Universal Robots PolyScope program: SandCube2.urp

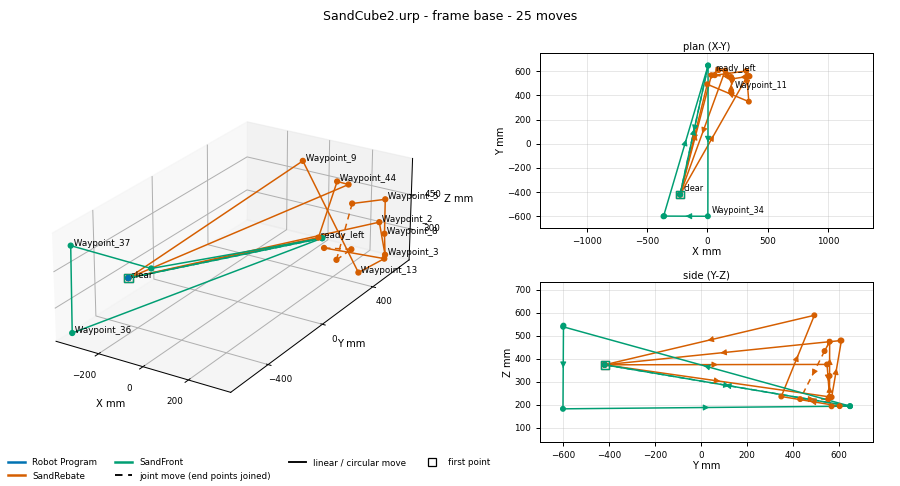
[picture p0: tool path of SandCube2.urp in frame base, 25 of 25 moves have a stored position in this frame; points joined in program order, loops and branches not executed]
Program SandCube2 (installation=main2 directory=/programs createdIn=5.11.5.1010327 lastSavedIn=5.11.5.1010327 robotSerialNumber=20215500677)
Calibrated DH parameters: a=[0.000204, -0.239222, -0.391845, -0.000001, 0.000022, 0]; d=[0.162722, -355.808559, 353.37206, 2.570385, 0.099741, 0.099629]; alpha=[1.571124, 0.000988, 0.008295, 1.568963, -1.570303, 0]; deltaTheta=[0, -0.973091, 7.204745, 0.05153, 0, 0]
Robot Program (runOnlyOnce=false)
  Folder Main
    MoveJ speed 60 deg/s, acceleration 80 deg/s^2 (useActiveTCP=false) tcp=DynabradeDual; feature=CubeFront
      Waypoint clear: TCP in base x=-225.713 y=-419.127 z=372.802 mm, rx=0.1834 ry=-2.2071 rz=2.1997 rad; joints [13.855, -106.476, 145.256, -123.976, 44.893, -104.552] deg; TCP offset x=3.18 y=114.64 z=98.2 mm, rx=-0.7854 ry=0 rz=0 rad; feature pose in base x=2.048 y=-607.004 z=173.227 mm, rx=-0.0204 ry=-2.2235 rz=-2.2094 rad
      URCap Zero FT Sensor (Robotiq_Copilot, Robotiq Inc.) dataModel(NodeInitializedKey=true, WaitForSteadyWrenchOptionKey=true)
    CubeFront := CubeFront
    Call SandFront
    CubeFront := SandBack
    Call SandFront
    SuppressedNode
      Call SprayFront
    SuppressedNode
      Call SprayFront
  SuppressedNode
    Folder Chamfer
      MoveL speed 250 mm/s, acceleration 1200 mm/s^2 (useActiveTCP=true) feature=Base
        MoveJ speed 60 deg/s, acceleration 80 deg/s^2 (useActiveTCP=true) feature=CubeFront
          Waypoint Waypoint_14: TCP in base x=40.557 y=344.633 z=644.318 mm, rx=1.3155 ry=-1.3725 rz=-1.2523 rad; joints [213.145, -95.792, 65.461, -31.373, -65.462, -328.995] deg; feature pose in base x=6.058 y=653.089 z=192.929 mm, rx=1.5716 ry=0.003 rz=-0.0025 rad
          Waypoint Waypoint_15: TCP in base x=-6.602 y=417.802 z=666.352 mm, rx=-2.8064 ry=0.3635 rz=0.257 rad; joints [242.083, -106.85, 75.59, -118.753, -70.655, -356.384] deg
          Waypoint Waypoint_16: TCP in base x=7.321 y=653.157 z=552.583 mm, rx=-2.3553 ry=0.0014 rz=0.0042 rad; joints [252.243, -84.14, 86.654, -182.715, -72.191, -359.211] deg
        URCap Find Surface (Robotiq_Copilot, Robotiq Inc.) dataModel(NodeInitializedKey=true, ZeroSensorBeforeKey=true, WaitForSteadyWrenchOptionKey=false, ls_force=10.0, ls_distance=100.0, ls_speed=5.0, ls_if_distance=false, ls_if_force=false); state(isChildrenLocked=true)
          'Add Stop conditions from the Find Surface node'
        URCap Finishing Tool Control (Robotiq_Copilot, Robotiq Inc.) dataModel(ToolOutputNameKey=digital_out[0], HackTriggeringContributionIsDefinedMethodKey=true)
        Wait Sleep waitTime=0.5
        MoveDirectionNode (selectedDirection=XPlus toolParams=0.15, 1.2) feature(featureName=CubeFront)
          Until DISTANCE (allowActions=false deceleration=3 distanceNodeType=STOP) Distance=0.35; motionParameters(blendRadius=0)
        MoveDirectionNode (selectedDirection=ZMinus) feature=Joint_6_name
          Until DISTANCE (allowActions=false deceleration=3 distanceNodeType=STOP) Distance=0.025; motionParameters(blendRadius=0)
        URCap Finishing Tool Control (Robotiq_Copilot, Robotiq Inc.) dataModel(FinishingToolStateKey=false, ToolOutputNameKey=digital_out[0], HackTriggeringContributionIsDefinedMethodKey=true)
        Waypoint Waypoint_18: TCP in base x=366.179 y=605.982 z=520.828 mm, rx=-1.6861 ry=0.1385 rz=1.2496 rad; joints [208.374, -44.818, 51.064, -237.69, -37.068, -253.683] deg
        URCap Find Surface (Robotiq_Copilot, Robotiq Inc.) dataModel(NodeInitializedKey=true, ZeroSensorBeforeKey=true, WaitForSteadyWrenchOptionKey=false, ls_force=10.0, ls_distance=100.0, ls_speed=5.0, ls_if_distance=false, ls_if_force=false); state(isChildrenLocked=true)
          'Add Stop conditions from the Find Surface node'
        URCap Finishing Tool Control (Robotiq_Copilot, Robotiq Inc.) dataModel(ToolOutputNameKey=digital_out[0], HackTriggeringContributionIsDefinedMethodKey=true)
        MoveDirectionNode (selectedDirection=YMinus toolParams=0.15, 1.2) feature(featureName=CubeFront)
          Until DISTANCE (allowActions=false deceleration=3 distanceNodeType=STOP) Distance=0.35; motionParameters(blendRadius=0)
        URCap Finishing Tool Control (Robotiq_Copilot, Robotiq Inc.) dataModel(FinishingToolStateKey=false, ToolOutputNameKey=digital_out[0], HackTriggeringContributionIsDefinedMethodKey=true)
        MoveDirectionNode (selectedDirection=ZMinus) feature=Joint_6_name
          Until DISTANCE (allowActions=false deceleration=3 distanceNodeType=STOP) Distance=0.05; motionParameters(blendRadius=0)
        Waypoint Waypoint_20: TCP in base x=366.722 y=626.869 z=194.22 mm, rx=-1.1174 ry=-0.6786 rz=-0.9417 rad; joints [212.764, -30.352, 68.609, -330.279, -35.41, -327.866] deg
        URCap Find Surface (Robotiq_Copilot, Robotiq Inc.) dataModel(NodeInitializedKey=true, ZeroSensorBeforeKey=true, WaitForSteadyWrenchOptionKey=false, ls_force=10.0, ls_distance=100.0, ls_speed=5.0, ls_if_distance=false, ls_if_force=false); state(isChildrenLocked=true)
          'Add Stop conditions from the Find Surface node'
        URCap Finishing Tool Control (Robotiq_Copilot, Robotiq Inc.) dataModel(ToolOutputNameKey=digital_out[0], HackTriggeringContributionIsDefinedMethodKey=true)
        Waypoint Waypoint_19: motionParameters(jointSpeed=1.047198 jointAcceleration=1.396263 cartesianSpeed=0.05 cartesianAcceleration=1.2); TCP in base x=29.784 y=640.794 z=212.679 mm, rx=-1.2502 ry=-0.1072 rz=-0.0765 rad; joints [247.483, -34.268, 98.117, -310.948, -74.468, -342.493] deg
        URCap Finishing Tool Control (Robotiq_Copilot, Robotiq Inc.) dataModel(FinishingToolStateKey=false, ToolOutputNameKey=digital_out[0], HackTriggeringContributionIsDefinedMethodKey=true)
        MoveDirectionNode (selectedDirection=ZMinus) feature=Joint_6_name
          Until DISTANCE (allowActions=false deceleration=3 distanceNodeType=STOP) Distance=0.05; motionParameters(blendRadius=0)
Event  expression=digital_in[1]≠ True
  Set DigitalOutput pin=digital_out[0]; digitalValue=0
  Set DigitalOutput pin=digital_out[1]; digitalValue=0
  Halt
SubProgram SandRebate (keepSynchronizedWithDisk=false)
  Folder sandRebate
    MoveJ speed 60 deg/s, acceleration 80 deg/s^2 (useActiveTCP=false) tcp=DynabradeDual; feature=CubeFront
      Waypoint clear: TCP in base x=-225.713 y=-419.127 z=372.802 mm, rx=0.1834 ry=-2.2071 rz=2.1997 rad; joints [13.855, -106.476, 145.256, -123.976, 44.893, -104.552] deg; feature pose in base x=2.048 y=-607.004 z=173.227 mm, rx=-0.0204 ry=-2.2235 rz=-2.2094 rad
      URCap Zero FT Sensor (Robotiq_Copilot, Robotiq Inc.) dataModel(NodeInitializedKey=true, WaitForSteadyWrenchOptionKey=true)
      MoveL speed 250 mm/s, acceleration 1200 mm/s^2 (useActiveTCP=false) tcp=DynabradeDual; feature=CubeFront
        Waypoint ready_left: TCP in base x=33.773 y=568.14 z=232.075 mm, rx=-1.2213 ry=-1.2022 rz=1.1979 rad; joints [233.005, -43.676, 101.374, -178.142, 55.004, -44.435] deg; TCP offset x=3.18 y=114.64 z=98.2 mm, rx=-0.7854 ry=0 rz=0 rad; feature pose in base x=9.685 y=618.378 z=176.869 mm, rx=1.5687 ry=-0.014 rz=-0.0074 rad
        URCap Find Surface (Robotiq_Copilot, Robotiq Inc.) dataModel(NodeInitializedKey=true, WaitForSteadyWrenchOptionKey=false, ls_force=10.0, ls_distance=100.0, ls_speed=5.0, ZeroSensorBeforeKey=true, ls_if_distance=false, ls_if_force=false); state(isChildrenLocked=true)
          'Add Stop conditions from the Find Surface node'
        URCap Finishing Tool Control (Robotiq_Copilot, Robotiq Inc.) dataModel(ToolOutputNameKey=digital_out[0], HackTriggeringContributionIsDefinedMethodKey=true)
        Wait Sleep waitTime=0.5
        Force Simple feature=Joint_6_name; selection=[0, 0, 1, 0, 0, 0]; wrench=[0, 0, 5, 0, 0, 0]; limitsForce=[0.15, 0.15, 0.15, 1.047198, 1.047198, 1.047198]; limitsMotion=[0.1, 0.1, 0.1, 0.349066, 0.349066, 0.349066]
          Waypoint Waypoint_44: motionParameters(jointSpeed=1.047198 jointAcceleration=1.396263 cartesianSpeed=0.05 cartesianAcceleration=1.2); TCP in base x=92.634 y=610.628 z=478.238 mm, rx=-0.8396 ry=-1.4025 rz=0.8393 rad; joints [232.816, -51.553, 73.036, -159.375, 69.035, -55.707] deg; TCP offset x=3.18 y=114.64 z=98.2 mm, rx=-0.7854 ry=0 rz=0 rad; feature pose in base x=85.344 y=655.608 z=190.328 mm, rx=1.5707 ry=0.001 rz=-0.0012 rad
        URCap Finishing Tool Control (Robotiq_Copilot, Robotiq Inc.) dataModel(ToolOutputNameKey=digital_out[0], HackTriggeringContributionIsDefinedMethodKey=true, FinishingToolStateKey=false)
        Waypoint Waypoint_4: TCP in base x=147.72 y=606.874 z=478.224 mm, rx=-0.8396 ry=-1.4025 rz=0.8394 rad; joints [229.161, -48.232, 67.407, -157.963, 71.791, -53.121] deg
        Waypoint clear: TCP in base x=-225.713 y=-419.127 z=372.802 mm, rx=0.1834 ry=-2.2071 rz=2.1997 rad; joints [13.855, -106.476, 145.256, -123.976, 44.893, -104.552] deg; feature pose in base x=2.048 y=-607.004 z=173.227 mm, rx=-0.0204 ry=-2.2235 rz=-2.2094 rad
        Waypoint Waypoint_2: TCP in base x=324.212 y=548.214 z=374.491 mm, rx=-1.2092 ry=1.2092 rz=-1.2092 rad; joints [245.591, -72.937, 106.11, -100.873, 130.52, -237.51] deg; feature pose in base x=6.058 y=653.089 z=192.929 mm, rx=1.5716 ry=0.003 rz=-0.0025 rad
        Waypoint Waypoint_3: TCP in base x=348.673 y=558.868 z=233.4 mm, rx=-1.199 ry=1.2125 rz=-1.2251 rad; joints [243.834, -57.283, 109.058, -119.037, 129.688, -236.76] deg; TCP offset x=3.18 y=114.64 z=98.2 mm, rx=-0.7854 ry=0 rz=0 rad; feature pose in base x=9.685 y=618.378 z=176.869 mm, rx=1.5687 ry=-0.014 rz=-0.0074 rad
        URCap Find Surface (Robotiq_Copilot, Robotiq Inc.) dataModel(NodeInitializedKey=true, WaitForSteadyWrenchOptionKey=false, ls_force=10.0, ls_distance=100.0, ls_speed=5.0, ZeroSensorBeforeKey=true, ls_if_distance=false, ls_if_force=false); state(isChildrenLocked=true)
          'Add Stop conditions from the Find Surface node'
        URCap Finishing Tool Control (Robotiq_Copilot, Robotiq Inc.) dataModel(ToolOutputNameKey=digital_out[0], HackTriggeringContributionIsDefinedMethodKey=true)
        Wait Sleep waitTime=0.5
        Force Simple feature=Joint_6_name; selection=[0, 0, 1, 0, 0, 0]; wrench=[0, 0, 5, 0, 0, 0]; limitsForce=[0.15, 0.15, 0.15, 1.047198, 1.047198, 1.047198]; limitsMotion=[0.1, 0.1, 0.1, 0.349066, 0.349066, 0.349066]
          Waypoint Waypoint_8: motionParameters(jointSpeed=1.047198 jointAcceleration=1.396263 cartesianSpeed=0.05 cartesianAcceleration=1.2); TCP in base x=343.269 y=559.127 z=324.456 mm, rx=2.2046 ry=-0.0122 rz=2.2215 rad; joints [241.547, -71.33, 93.008, -21.809, 107.451, -270.149] deg; TCP offset x=3.18 y=114.64 z=98.2 mm, rx=-0.7854 ry=0 rz=0 rad
          Waypoint Waypoint_5: motionParameters(jointSpeed=1.047198 jointAcceleration=1.396263 cartesianSpeed=0.05 cartesianAcceleration=1.2); TCP in base x=342.13 y=559.447 z=473.527 mm, rx=2.1002 ry=0.2016 rz=2.1132 rad; joints [241.727, -73.096, 71.489, 10.077, 107.843, -275.731] deg; TCP offset x=3.18 y=114.64 z=98.2 mm, rx=-0.7854 ry=0 rz=0 rad
        URCap Finishing Tool Control (Robotiq_Copilot, Robotiq Inc.) dataModel(FinishingToolStateKey=false, ToolOutputNameKey=digital_out[0], HackTriggeringContributionIsDefinedMethodKey=true)
        Waypoint Waypoint_17: TCP in base x=204.615 y=537.314 z=432.533 mm, rx=-1.1836 ry=-1.1482 rz=-1.3158 rad; joints [212.134, -87.867, 98.846, 1.992, -9.504, -287.219] deg; TCP offset x=3.18 y=114.64 z=98.2 mm, rx=-0.7854 ry=0 rz=0 rad; feature pose in base x=6.058 y=653.089 z=192.929 mm, rx=1.5716 ry=0.003 rz=-0.0025 rad
        MoveJ speed 60 deg/s, acceleration 80 deg/s^2 (useActiveTCP=true) feature=CubeFront
          Waypoint Waypoint_11: TCP in base x=197.023 y=431.256 z=223.624 mm, rx=2.362 ry=2.0713 rz=0 rad; joints [223.025, -89.028, 102.064, -70.501, -56.519, -139.472] deg
          Waypoint Waypoint_6: TCP in base x=196.959 y=553.123 z=223.756 mm, rx=-1.75 ry=-2.609 rz=-0.0001 rad; joints [233.913, -69.804, 77.285, -56.958, -67.897, -156.703] deg
          Waypoint Waypoint_31: TCP in base x=61.467 y=567.687 z=192.19 mm, rx=1.7638 ry=2.5902 rz=0.0029 rad; joints [245.976, -73.297, 87.687, -68.963, -60.284, -145.062] deg; TCP offset x=3.18 y=114.64 z=98.2 mm, rx=-0.7854 ry=0 rz=0 rad; feature pose in base x=9.685 y=618.378 z=176.869 mm, rx=1.5687 ry=-0.014 rz=-0.0074 rad
          URCap Zero FT Sensor (Robotiq_Copilot, Robotiq Inc.) dataModel(NodeInitializedKey=true, WaitForSteadyWrenchOptionKey=true)
        URCap Find Surface (Robotiq_Copilot, Robotiq Inc.) dataModel(NodeInitializedKey=true, ZeroSensorBeforeKey=true, WaitForSteadyWrenchOptionKey=false, ls_force=10.0, ls_distance=100.0, ls_speed=5.0, ls_if_distance=false, ls_if_force=false); state(isChildrenLocked=true)
          'Add Stop conditions from the Find Surface node'
        URCap Finishing Tool Control (Robotiq_Copilot, Robotiq Inc.) dataModel(ToolOutputNameKey=digital_out[0], HackTriggeringContributionIsDefinedMethodKey=true)
        Wait Sleep waitTime=0.5
        Force Frame feature=Joint_6_name; selection=[0, 0, 1, 0, 0, 0]; wrench=[0, 0, 5, 0, 0, 0]; limitsForce=[0.15, 0.15, 0.15, 1.047198, 1.047198, 1.047198]; limitsMotion=[0.1, 0.1, 0.1, 0.349066, 0.349066, 0.349066]
          Waypoint Waypoint_7: motionParameters(jointSpeed=1.047198 jointAcceleration=1.396263 cartesianSpeed=0.05 cartesianAcceleration=1.2); TCP in base x=322.305 y=603.203 z=193.01 mm, rx=2.5491 ry=1.8349 rz=-0.0035 rad; joints [225.958, -61.111, 72.887, -78.246, -49.944, -124.133] deg; TCP offset x=3.18 y=114.64 z=98.2 mm, rx=-0.7854 ry=0 rz=0 rad; feature pose in base x=6.058 y=653.089 z=192.929 mm, rx=1.5716 ry=0.003 rz=-0.0025 rad
        URCap Finishing Tool Control (Robotiq_Copilot, Robotiq Inc.) dataModel(FinishingToolStateKey=false, ToolOutputNameKey=digital_out[0], HackTriggeringContributionIsDefinedMethodKey=true)
        Waypoint Waypoint_13: TCP in base x=343.245 y=349.195 z=234.967 mm, rx=-1.8514 ry=-2.5381 rz=0.0001 rad; joints [208.052, -81.166, 89.339, -53.576, -82.434, -172.912] deg; feature pose in base x=9.685 y=618.378 z=176.869 mm, rx=1.5687 ry=-0.014 rz=-0.0074 rad
        Waypoint Waypoint_9: TCP in base x=-0.811 y=492.962 z=588.061 mm, rx=-1.9827 ry=-0.1778 rz=-0.0774 rad; joints [237.765, -113.533, 89.133, -2.101, 52.621, -171.272] deg
        Waypoint clear: TCP in base x=-225.713 y=-419.127 z=372.802 mm, rx=0.1834 ry=-2.2071 rz=2.1997 rad; joints [13.855, -106.476, 145.256, -123.976, 44.893, -104.552] deg; feature pose in base x=2.048 y=-607.004 z=173.227 mm, rx=-0.0204 ry=-2.2235 rz=-2.2094 rad
SubProgram  [hidden by the author, left out]
SubProgram SprayRebate [hidden by the author, left out]
SubProgram -> SandFront
SubProgram StartSpray [hidden by the author, left out]
SubProgram stopSpray [hidden by the author, left out]
SubProgram SandFront (keepSynchronizedWithDisk=false)
  Folder sandFront
    MoveJ speed 60 deg/s, acceleration 80 deg/s^2 (useActiveTCP=false) tcp=DynabradeDual; feature=CubeFront
      Waypoint clear: TCP in base x=-225.713 y=-419.127 z=372.802 mm, rx=0.1834 ry=-2.2071 rz=2.1997 rad; joints [13.855, -106.476, 145.256, -123.976, 44.893, -104.552] deg
    MoveL speed 250 mm/s, acceleration 1200 mm/s^2 (useActiveTCP=false) tcp=DynabradeDual; feature=CubeFront
      Waypoint Waypoint_1: TCP in base x=6.072 y=648.1 z=192.982 mm, rx=-1.5699 ry=0.0092 rz=0.0097 rad; joints [251.403, -67.593, 131.535, -110.394, 77.851, -166.352] deg; feature pose in base x=6.058 y=653.089 z=192.929 mm, rx=1.5716 ry=0.003 rz=-0.0025 rad
      URCap Zero FT Sensor (Robotiq_Copilot, Robotiq Inc.) dataModel(NodeInitializedKey=true, WaitForSteadyWrenchOptionKey=true)
      URCap Find Surface (Robotiq_Copilot, Robotiq Inc.) dataModel(NodeInitializedKey=true, WaitForSteadyWrenchOptionKey=false, ls_force=10.0, ls_distance=100.0, ls_speed=5.0, ZeroSensorBeforeKey=false, ls_if_distance=false, ls_if_force=false); state(isChildrenLocked=true)
        'Add Stop conditions from the Find Surface node'
      URCap Finishing Tool Control (Robotiq_Copilot, Robotiq Inc.) dataModel(ToolOutputNameKey=digital_out[0], HackTriggeringContributionIsDefinedMethodKey=true)
      Wait Sleep waitTime=0.5
    MoveL speed 60 mm/s, acceleration 1200 mm/s^2 (useActiveTCP=false) tcp=DynabradeDual; feature=CubeFront
      Force Simple feature=Joint_6_name; selection=[0, 0, 1, 0, 0, 0]; wrench=[0, 0, 5, 0, 0, 0]; limitsForce=[0.15, 0.15, 0.15, 1.047198, 1.047198, 1.047198]; limitsMotion=[0.1, 0.1, 0.1, 0.349066, 0.349066, 0.349066]
        Waypoint Waypoint_34: TCP in base x=4.168 y=-599.662 z=538.228 mm, rx=0.1003 ry=-2.1628 rz=2.1762 rad; joints [69.8, -105.08, 109.114, -52.157, 72.617, -168.988] deg; feature pose in base x=2.048 y=-607.004 z=173.227 mm, rx=-0.0204 ry=-2.2235 rz=-2.2094 rad
        Waypoint Waypoint_37: TCP in base x=-357.721 y=-598.101 z=543.274 mm, rx=0.1002 ry=-2.1629 rz=2.1762 rad; joints [31.577, -86.57, 95.791, -75.508, 51.138, -132.637] deg
        Waypoint Waypoint_36: TCP in base x=-362.939 y=-600.337 z=181.342 mm, rx=0.1002 ry=-2.1628 rz=2.1761 rad; joints [31.404, -55.313, 118.507, -129.285, 51.013, -132.956] deg
        Waypoint Waypoint_1: TCP in base x=6.072 y=648.1 z=192.982 mm, rx=-1.5699 ry=0.0092 rz=0.0097 rad; joints [251.403, -67.593, 131.535, -110.394, 77.851, -166.352] deg; feature pose in base x=6.058 y=653.089 z=192.929 mm, rx=1.5716 ry=0.003 rz=-0.0025 rad
        URCap Finishing Tool Control (Robotiq_Copilot, Robotiq Inc.) dataModel(FinishingToolStateKey=false, ToolOutputNameKey=digital_out[0], HackTriggeringContributionIsDefinedMethodKey=true)
      MoveDirectionNode (selectedDirection=ZMinus) feature=Joint_6_name
        Until DISTANCE (allowActions=false deceleration=3 distanceNodeType=STOP) Distance=0.025; motionParameters(blendRadius=0)
    MoveJ speed 60 deg/s, acceleration 80 deg/s^2 (useActiveTCP=true) feature=CubeFront
      Waypoint clear: TCP in base x=-225.713 y=-419.127 z=372.802 mm, rx=0.1834 ry=-2.2071 rz=2.1997 rad; joints [13.855, -106.476, 145.256, -123.976, 44.893, -104.552] deg; feature pose in base x=2.048 y=-607.004 z=173.227 mm, rx=-0.0204 ry=-2.2235 rz=-2.2094 rad
SubProgram SprayFront [hidden by the author, left out]
